(* PLC project SafeLOGIC-1, BrAutomation SafeDESIGNER  5.15.0.0 *)
(* stored: companyURL http://www.br-automation.com, creationDateTime Thu Jan 06 16:36:38 2022 *)

PROGRAM Output

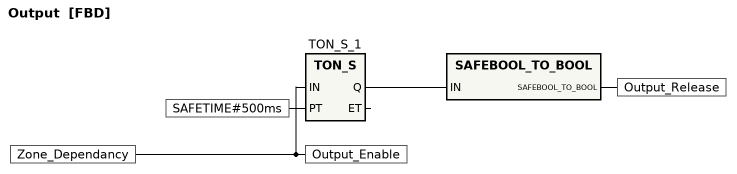
(* FBD diagram, written out as Structured Text *)
Output_Enable := Zone_Dependancy;
TON_S_1(IN := Zone_Dependancy, PT := SAFETIME#500ms);
Output_Release := SAFEBOOL_TO_BOOL(TON_S_1.Q);
END_PROGRAM
